Yaskawa INFORM job: TEST-OS-X.JBI

/JOB
//NAME TEST-OS-X
//POS
///NPOS 2,2,0,0,0,0
///TOOL 0
///POSTYPE PULSE
///PULSE
C00000=6100,8040,48141,-69136,105320,27890
C00001=6100,8040,48142,-69136,105320,27891
BC00000=22318,663670,413407
BC00001=368028,663671,413407
//INST
///DATE 2025/04/16 15:51
///ATTR SC,RW
///GROUP1 RB1,BS1
NOP
*LABEL
MOVJ C00000 BC00000 VJ=80.00
MOVJ C00001 BC00001 VJ=80.00
JUMP *LABEL
END
